FUNCTION_BLOCK TableLogic
VAR
	timer: TOF;
	timerElapsed: BOOL;
	riseTrig: R_TRIG;
	riseTrigDetected: BOOL;
	counter: CTU;
	trigerForTriger: bool;
	timer2: TOF;
	timer2elapsed: bool;
	trigerForTriger2: bool;
	delay: TON;
END_VAR

riseTrig(CLK := gvl.SwitchPress, Q => riseTrigDetected);
timer(IN := riseTrigDetected, PT := LocalVariables.Recipe.WorkingTime, Q => timerElapsed);

gvl.MotorTableMove := TRUE;

IF riseTrigDetected THEN
	LocalVariables.Locations[3].Item.Id := LocalVariables.Locations[2].Item.Id;
	LocalVariables.Locations[3].Item.Recipe := LocalVariables.Locations[2].Item.Recipe;
	LocalVariables.Locations[2].Item.Id := 0;
	LocalVariables.Locations[2].Item.Recipe := LocalVariables.Recipe;
END_IF

IF timerElapsed THEN
	gvl.PistonPress := TRUE;
	gvl.MotorTableMove := FALSE;
ELSIF NOT gvl.FotocellOutput THEN
	gvl.MotorTableMove := FALSE;
	gvl.PistonPress := FALSE;
ELSE	
	gvl.PistonPress := FALSE;
	gvl.MotorTableMove := TRUE;
END_IF

END_FUNCTION_BLOCK

(* stored: Version 1.1.0.1, ProductVersion 3.1.4024.12
   POU TableLogic: Id {f635f7ab-4fc0-4104-8ada-04baa1f4a91b}, SpecialFunc None *)
